TYPE Error :
STRUCT
	Active : BOOL; // TRUE = error is active
	Code : INT; // Error return code => E_ErrorCode
	Info : Tc2_System.T_MaxString; // Error message
END_STRUCT
END_TYPE

(* stored: Version 1.1.0.1
   DUT Error: Id {23c996c0-f051-4322-bcdc-8cc9475229f8} *)
